{attribute 'linkalways'} 
{attribute 'no_explicit_call' := 'This FB is a CLASS and must be accessed using methods or properties'}
{attribute 'enable_dynamic_creation'}
FUNCTION_BLOCK _ETcVnLineType EXTENDS EnumDatatypeBase
VAR
	localData : ETcVnLineType;
	activeData : REFERENCE TO ETcVnLineType;
	enumBaseDatatype : _DINT(localData);
END_VAR

METHOD PRIVATE AddLocalEnumeration
VAR_INPUT
	Enumeration : T_MAXSTRING;
	Value : ETcVnLineType;
END_VAR
AddEnumeration(Enumeration, Value);
END_METHOD

PROPERTY PUBLIC Address : PVOID
GET
Address := ADR(activeData);
END_GET
END_PROPERTY

METHOD PUBLIC ClearReference
VAR_INPUT
END_VAR
activeData REF= localData;
SetBaseDatatypeReference();
END_METHOD

METHOD PUBLIC Clone : I_Datatype
VAR
    pClone : POINTER TO _ETcVnLineType;
END_VAR
pClone := __NEW(_ETcVnLineType(InitialValue := Value));
Clone := pClone^;
END_METHOD

METHOD FB_init : BOOL
VAR_INPUT
	bInitRetains : BOOL; // if TRUE, the retain variables are initialized (warm start / cold start)
	bInCopyCode : BOOL;  // if TRUE, the instance afterwards gets moved into the copy code (online change)
	InitialValue : ETcVnLineType;
END_VAR
localData := InitialValue;
AddBaseDatatype(enumBaseDatatype);
ClearReference();

AddLocalEnumeration('TCVN_LT_4_CONNECTED', ETcVnLineType.TCVN_LT_4_CONNECTED);
AddLocalEnumeration('TCVN_LT_8_CONNECTED', ETcVnLineType.TCVN_LT_8_CONNECTED);
AddLocalEnumeration('TCVN_LT_ANTIALIASED', ETcVnLineType.TCVN_LT_ANTIALIASED);
END_METHOD

PROPERTY PUBLIC Identifier : T_MAXSTRING
GET
Identifier := 'ETcVnLineType';
END_GET
END_PROPERTY

METHOD IsEnumeratorValueEqual : BOOL
VAR_INPUT
	Enumerator : I_KeyValueForwardEnumerator;
END_VAR
VAR
	storedValue : ETcVnLineType;
END_VAR
IF NOT Enumerator.TryGet(storedValue) THEN
	RETURN;
END_IF

IsEnumeratorValueEqual := storedValue = activeData;
END_METHOD

METHOD PUBLIC MakeReferenceTo
VAR_INPUT
	ReferenceTarget : REFERENCE TO ETcVnLineType;
END_VAR
activeData REF= ReferenceTarget;
SetBaseDatatypeReference();
END_METHOD

METHOD PROTECTED SetBaseDatatypeReference
VAR_INPUT
END_VAR
enumBaseDatatype.MakeReferenceTo(activeData);
END_METHOD

PROPERTY PUBLIC Size : UDINT
GET
Size := SIZEOF(activeData);
END_GET
END_PROPERTY

METHOD TryMakeReferenceTo : BOOL
VAR_INPUT
	Target : I_Datatype;
END_VAR
VAR
	targetAsEnum : I_EnumDatatype;
	pTargetData : POINTER TO ETcVnLineType;
END_VAR
IF NOT Target.TryResolveAsEnumDatatype(targetAsEnum) THEN
	RETURN;
END_IF

IF targetAsEnum.Identifier <> Identifier THEN
	RETURN;
END_IF

pTargetData := Target.Address;
activeData REF= pTargetData^;
SetBaseDatatypeReference();
TryMakeReferenceTo := TRUE;
END_METHOD

PROPERTY PUBLIC Value : ETcVnLineType
GET
Value := activeData;
END_GET
SET
activeData := Value;
END_SET
END_PROPERTY

END_FUNCTION_BLOCK

(* stored: Version 1.1.0.1, ProductVersion 3.1.4024.12
   POU _ETcVnLineType: Id {3920339e-3478-0939-28a5-9b9235d595cf}, SpecialFunc None
   Folder Constructor: Id {f3fc32b5-a1c2-0b42-32fe-a90d0145395c}
   Folder Private: Id {63731e52-8e40-0ecc-12ad-44355a624eeb}
   Folder Protected: Id {56af0d7b-0b55-04fb-131e-cef5272c44eb}
   Method AddLocalEnumeration: Id {f257eaab-208c-013e-1f64-547722f47a74}
   Property Address: Id {e98658a4-d241-0706-3690-364a3a2657b0}
   Get Get: Id {dad46421-692c-0c98-2887-49efad423870}
   Method ClearReference: Id {7310b07c-2c63-0046-1c7d-8f27d25eb75e}
   Method Clone: Id {5864c546-3b9f-0097-1430-b33dd2f6d040}
   Method FB_init: Id {26ce0258-c308-09ab-04ec-f725ff644b6a}
   Property Identifier: Id {85d07dbb-6161-0b28-3c69-e66877138447}
   Get Get: Id {b644d78c-5d41-0841-3192-7acced11041c}
   Method IsEnumeratorValueEqual: Id {2f49cfb8-3957-0c9d-3312-bcb74db0d3ba}
   Method MakeReferenceTo: Id {f7ea204c-44cd-0d14-09ca-60d86e10cbc7}
   Method SetBaseDatatypeReference: Id {5f6a6758-465f-0cf1-3a80-0b22132bc966}
   Property Size: Id {328d68b1-b9f8-06bc-37aa-27b79f78c3e6}
   Get Get: Id {373fc034-8ad3-059c-181b-b90cd1981c15}
   Method TryMakeReferenceTo: Id {cc84f1d9-ec7a-09d9-1b93-a00188288c00}
   Property Value: Id {aaac26db-e216-02cc-2949-12f7e7836354}
   Get Get: Id {cb95fc19-f733-075f-3ed1-3293911ac2bd}
   Set Set: Id {daa82ede-cc20-08eb-3975-867452603ee0} *)
